// TIA Portal V16 export
// export: Created 2022-11-17T11:55:29.9296508Z, ExportSetting WithDefaults, DisplayName Totally Integrated Automation Portal, DisplayVersion V16 Update 6, DisplayName TIA Portal Version Control Interface, DisplayVersion V16 Update 2, DisplayName TIA Portal Openness, DisplayVersion V16 Update 6, DisplayName SINAMICS Startdrive Advanced, DisplayVersion V16 Update 5, DisplayName SINAMICS Startdrive G130, G150, S120, S150, SINAMICS MV, S210, DisplayVersion V16 Update 5, DisplayName SINAMICS Startdrive G110M, G120, G120C, G120D, G120P, G115D, DisplayVersion V16 Update 5, DisplayName STEP 7 Professional, DisplayVersion V16 Update 6, DisplayName STEP 7 Safety, DisplayVersion V16, DisplayName WinCC Advanced, DisplayVersion V16 Update 6
DATA_BLOCK "DB80_Label"   // DB80
{ S7_Optimized_Access := 'FALSE' }
VERSION : 0.1
// stored: AutoNumber false, IsOnlyStoredInLoadMemory false, IsWriteProtectedInAS false
   VAR RETAIN
      Step0 : Bool := FALSE;   // Table rotation to first label position
      Step1 : Bool := FALSE;   // First label apply
      Step2 : Bool := FALSE;   // Table rotation to second label position
      Step3 : Bool := FALSE;   // Second label apply
      Step4 : Bool := FALSE;   // Table rotation to third label position
      Step5 : Bool := FALSE;   // Third label apply
      Step6 : Bool := FALSE;   // Table rotation to fourth label position
      Step7 : Bool := FALSE;   // Fourt label apply
      Step8 : Bool := FALSE;   // Table rotation to end cycle position
      spare_Step9 : Bool := FALSE;
      spare_Step10 : Bool := FALSE;
      spare_Step11 : Bool := FALSE;
      spare_Step12 : Bool := FALSE;
      spare_Step13 : Bool := FALSE;
      spare_Step14 : Bool := FALSE;
      spare_Step15 : Bool := FALSE;
      Phase1_On : Bool := TRUE;
      Phase2_On : Bool := FALSE;
      Phase3_On : Bool := TRUE;
      Phase4_On : Bool := FALSE;
      Enable : Bool := TRUE;
      rotation : Bool := FALSE;   // Table rotation for label command
      label_ok1 : Bool := FALSE;   // Label cycle ended
      S1 : Bool := FALSE;   // Label request signal
      spare_signal2 : Bool := FALSE;
      spare_signal3 : Bool := FALSE;
      spare_signal4 : Bool := FALSE;
      spare_signal5 : Bool := FALSE;
      spare_signal6 : Bool := FALSE;
      spare_signal7 : Bool := FALSE;
      spare_signal8 : Bool := FALSE;
      E1 : Bool := TRUE;   // Label arm in home position for pallet transit
      E2 : Bool := FALSE;   // Label applied signal
      E3 : Bool := FALSE;   // Label fault signal
      spare_input4 : Bool := FALSE;
      spare_input5 : Bool := FALSE;
      spare_input6 : Bool := FALSE;
      spare_input7 : Bool := FALSE;
      spare_input8 : Bool := FALSE;
      spare_byte5 : Byte := 16#00;
      Phase1 : Int := 900;
      Phase2 : Int := 1800;
      Phase3 : Int := 2700;
      Phase4 : Int := 3600;
      NextPhase : Int := 2700;
   END_VAR
BEGIN
END_DATA_BLOCK
